Fanuc KAREL source: kt00737.KL

-- PROVISIONAL review KL for V770-1; original PC SHA256 091e69cc2c2ff737e94fbd0e0bb8223761f14bcd15f13155ac35a70fc7299f5b
-- Incomplete behavior may be omitted. Consult companion uncertainty JSON. Do not deploy.
PROGRAM KT00737
%NOLOCKGROUP
BEGIN
  -- UNRESOLVED_PC offsets 5-18; opcodes 22,1D,23
  -- UNRESOLVED_PC offsets 23-27; opcodes 7F
END KT00737
